{attribute 'qualified_only'}
VAR_GLOBAL
	K1	 AT %Q*:BOOL;     // 	Ventil Zylinder ausfahren
	K2	 AT %Q*:BOOL;     // 	Ventil Zylinder einfahren
	P1	 AT %Q*:BOOL;     // 	Meldeleuchte Betriebsbereit
	P2	 AT %Q*:BOOL;     // 	Meldeleuchte Sammelstörung
	P3	 AT %Q*:BOOL;     // 	Meldeleuchte STörung Motor
	P4	 AT %Q*:BOOL;     // 	Meldeleuchte Überdruck
	P5	 AT %Q*:BOOL;     // 	Meldeleuchte Druck erreicht
	P6	 AT %Q*:BOOL;     // 	Meldeleuchte Ölstand MIN.
	P7	 AT %Q*:BOOL;     // 	Meldeleuchte Lüfter Ölkühler
	P8	 AT %Q*:BOOL;     // 	Meldeleuchte Ölfilter wechseln
	Q1	 AT %Q*:BOOL;     // 	Netzschütz
	Q2	 AT %Q*:BOOL;     // 	Sternschütz
	Q3	 AT %Q*:BOOL;     // 	Dreieckschütz
	Q4	 AT %Q*:BOOL;     // 	Lüfter Ölkühler
END_VAR

(* stored: Version 1.1.0.1, ProductVersion 3.1.4024.5
   GVL DA: Id {efa3d63a-96e1-4204-b1e7-9f3703bd4f03} *)
